// TIA Portal V17 export
// export: Created 2022-10-14T12:26:28.7230279Z, ExportSetting WithDefaults, DisplayName Totally Integrated Automation Portal, DisplayVersion V17 Update 4, DisplayName TIA Portal Openness, DisplayVersion V17 Update 4, DisplayName TIA Portal Version Control Interface, DisplayVersion V17, DisplayName SINAMICS Startdrive Advanced, DisplayVersion V17 Update2, DisplayName SINAMICS Startdrive G130, G150, S120, S150, SINAMICS MV, S210, DisplayVersion V17 Update2, DisplayName SINAMICS Startdrive G110M, G120, G120C, G120D, G120P, G115D, DisplayVersion V17 Update2, DisplayName STEP 7 Professional, DisplayVersion V17 Update 4, DisplayName STEP 7 Safety, DisplayVersion V17, DisplayName WinCC Advanced / Unified PC, DisplayVersion V17 Update 4
FUNCTION "REAL_Anzeige" : Void   // FC2, FBD
{ S7_Optimized_Access := 'TRUE' }
VERSION : 0.1
// stored: AutoNumber true, IsIECCheckEnabled false, SetENOAutomatically false, UDAEnableTagReadback false
   VAR_INPUT
      IN_Real : Real;
   END_VAR
   VAR_OUTPUT
      Anzeige_1 : Int;
      Anzeige_2 : Int;
      Anzeige_3 : Int;
   END_VAR
   VAR_TEMP
      HBcd_0 : Word;
      HBcd_1 : Word;
      HInt_0 : Int;
      HInt_1 : Int;
      HInt_2 : Int;
      Hint_3 : Int;
      HReal_0 : Real;
      HReal_1 : Real;
      HReal_2 : Real;
      HReal_3 : Real;
      HReal_4 : Real;
      HReal_5 : Real;
      ABS_Real : Real;
   END_VAR
BEGIN

REGION Network 1
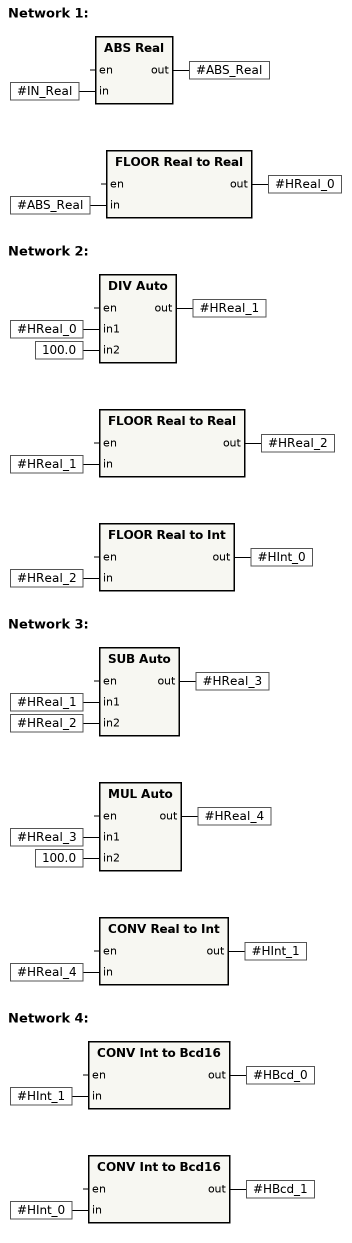
   #ABS_Real := ABS(#IN_Real);
   #HReal_0 := FLOOR(#ABS_Real);
END_REGION

REGION Network 2
   #HReal_1 := #HReal_0 / 100.0;
   #HReal_2 := FLOOR(#HReal_1);
   #HInt_0 := FLOOR(#HReal_2);
END_REGION

REGION Network 3
   #HReal_3 := #HReal_1 - #HReal_2;
   #HReal_4 := #HReal_3 * 100.0;
   #HInt_1 := REAL_TO_INT(#HReal_4);
END_REGION

REGION Network 4
   #HBcd_0 := INT_TO_BCD16(#HInt_1);
   #HBcd_1 := INT_TO_BCD16(#HInt_0);
END_REGION

REGION Network 5
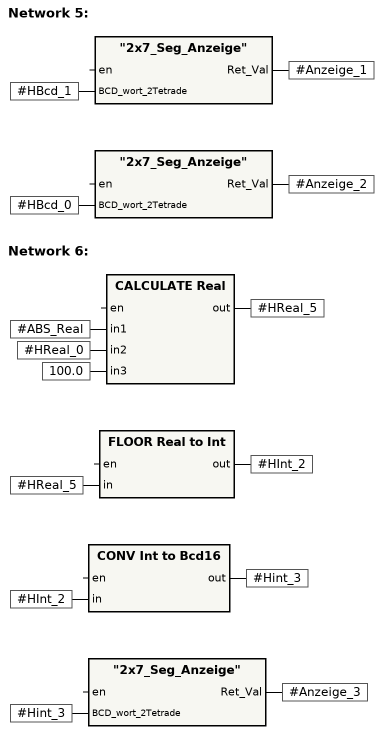
   #Anzeige_1 := "2x7_Seg_Anzeige"(BCD_wort_2Tetrade := #HBcd_1);
   #Anzeige_2 := "2x7_Seg_Anzeige"(BCD_wort_2Tetrade := #HBcd_0);
END_REGION

REGION Network 6
   #HReal_5 := (#ABS_Real-#HReal_0)*100.0;
   #HInt_2 := FLOOR(#HReal_5);
   #Hint_3 := INT_TO_BCD16(#HInt_2);
   #Anzeige_3 := "2x7_Seg_Anzeige"(BCD_wort_2Tetrade := #Hint_3);
END_REGION
END_FUNCTION
